FUNCTION_BLOCK DrillingActuatorVertical EXTENDS ZEquipment.ActuatorDigitalBiLsPlusMinus

METHOD PUBLIC AufAsync
VAR_INPUT
  startToken : ZCore.IStartToken;
END_VAR
MovePlusAsync(startToken:=startToken);
END_METHOD

METHOD PUBLIC Geschlossen : BOOL
VAR_INPUT
END_VAR
Geschlossen := IsAtMinus();
END_METHOD

METHOD PUBLIC Offen : BOOL
VAR_INPUT
END_VAR
Offen := IsAtPlus();
END_METHOD

METHOD PUBLIC ZuAsync
VAR_INPUT
  startToken : ZCore.IStartToken;
END_VAR
MoveMinusAsync(startToken:=startToken);
END_METHOD

END_FUNCTION_BLOCK

(* stored: Version 1.1.0.1
   POU DrillingActuatorVertical: Id {eb570af9-9080-41f8-81d4-a1210ee34018}, SpecialFunc None
   Method AufAsync: Id {3efd8727-d9fd-423e-b6c3-bba8087507f6}
   Method Geschlossen: Id {4c473d52-84a7-4e51-8dc4-09552c9cce3b}
   Method Offen: Id {d0e43d0e-7883-4d4f-a1fb-faa4c0c21c14}
   Method ZuAsync: Id {aad59b46-816a-4129-b948-f99a915de6a9} *)
